SUBAPPLICATION Uebung_072c_AUI (* GBSD und WBSD auf UT ausgeben mit PHYS (Adapter Version) *)
  (* Standard: 61499-2; Description: Copyright (c) 2023 Meisterschulen am Ostbahnhof This program and the accompanying materials are made available under the terms of the Eclipse Public License 2.0 which is available at https://www.eclipse.org/legal/epl-2.0/ SPDX-License-Identifier: EPL-2.0 *)
  (* Version 1.0, 2026-06-01, Franz Höpfinger, Meisterschulen am Ostbahnhof, GBSD und WBSD mit PHYS Skalierung (Adapter Version) *)
  PACKAGE Uebungen;
  IMPORT Uebungen::const::UT::TECU::DefaultPool_TECU_Numeric::NumberVariable_Ground_based_machine_speed_N;
  IMPORT Uebungen::const::UT::TECU::DefaultPool_TECU_Numeric::NumberVariable_Wheel_based_machine_speed_N;
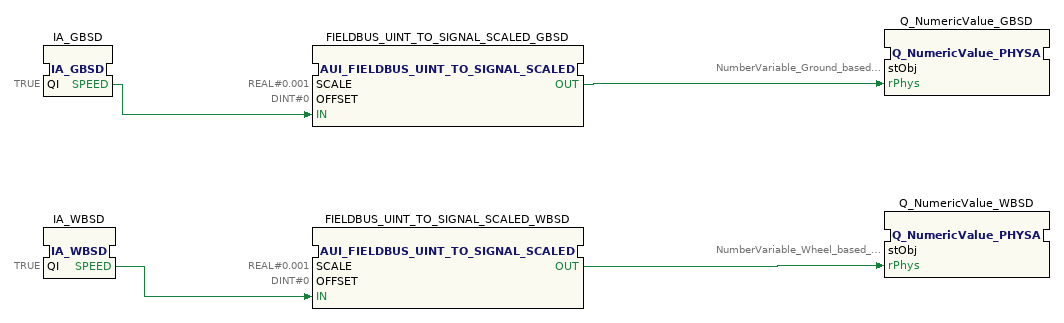
  FBS
    IA_GBSD : isobus::tecu::IA_GBSD(QI := TRUE);
    IA_WBSD : isobus::tecu::IA_WBSD(QI := TRUE);
    FIELDBUS_UINT_TO_SIGNAL_SCALED_GBSD : logiBUS::signalprocessing::fieldbus::AUI_FIELDBUS_UINT_TO_SIGNAL_SCALED(SCALE := REAL#0.001, OFFSET := DINT#0);
    FIELDBUS_UINT_TO_SIGNAL_SCALED_WBSD : logiBUS::signalprocessing::fieldbus::AUI_FIELDBUS_UINT_TO_SIGNAL_SCALED(SCALE := REAL#0.001, OFFSET := DINT#0);
    Q_NumericValue_GBSD : isobus::UT::Q::Q_NumericValue_PHYSA(stObj := NumberVariable_Ground_based_machine_speed_N);
    Q_NumericValue_WBSD : isobus::UT::Q::Q_NumericValue_PHYSA(stObj := NumberVariable_Wheel_based_machine_speed_N);
  END_FBS
  ADAPTER_CONNECTIONS
    IA_GBSD.SPEED TO FIELDBUS_UINT_TO_SIGNAL_SCALED_GBSD.IN;
    FIELDBUS_UINT_TO_SIGNAL_SCALED_GBSD.OUT TO Q_NumericValue_GBSD.rPhys;
    IA_WBSD.SPEED TO FIELDBUS_UINT_TO_SIGNAL_SCALED_WBSD.IN;
    FIELDBUS_UINT_TO_SIGNAL_SCALED_WBSD.OUT TO Q_NumericValue_WBSD.rPhys;
  END_CONNECTIONS
END_SUBAPPLICATION
